// Mitsubishi GX Works2 project: TEACH 실습 예제   PLC: Q03UDV

PROGRAM MAIN
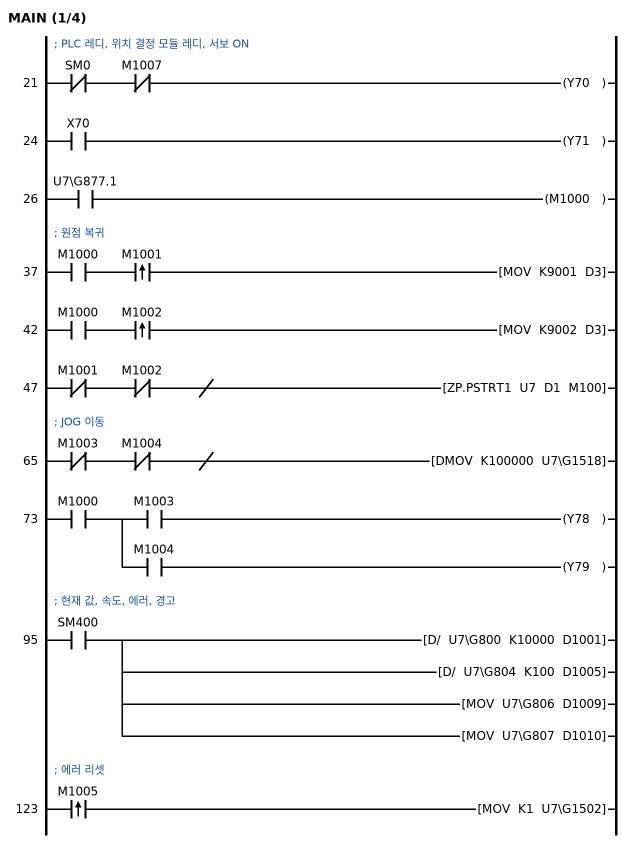
; PLC 레디, 위치 결정 모듈 레디, 서보 ON
21    LDI     SM0
      ANI     M1007
      OUT     Y70
24    LD      X70
      OUT     Y71
26    LD      U7\G877.1
      OUT     M1000
; 원점 복귀
37    LD      M1000
      ANDP    M1001
      MOV     K9001 D3
42    LD      M1000
      ANDP    M1002
      MOV     K9002 D3
47    LDI     M1001
      ANI     M1002
      INV
      ZP.PSTRT1 U7 D1 M100
; JOG 이동
65    LDI     M1003
      ANI     M1004
      INV
      DMOV    K100000 U7\G1518
73    LD      M1000
      MPS
      AND     M1003
      OUT     Y78
      MPP
      AND     M1004
      OUT     Y79
; 현재 값, 속도, 에러, 경고
95    LD      SM400
      D/      U7\G800 K10000 D1001
      D/      U7\G804 K100 D1005
      MOV     U7\G806 D1009
      MOV     U7\G807 D1010
; 에러 리셋
123   LDP     M1005
      MOV     K1 U7\G1502
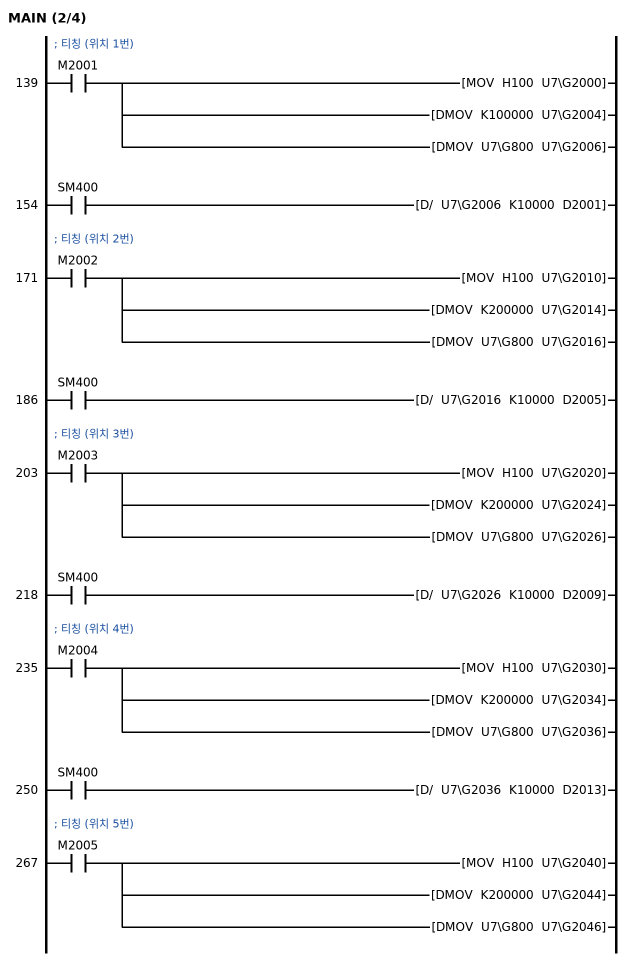
; 티칭 (위치 1번)
139   LD      M2001
      MOV     H100 U7\G2000
      DMOV    K100000 U7\G2004
      DMOV    U7\G800 U7\G2006
154   LD      SM400
      D/      U7\G2006 K10000 D2001
; 티칭 (위치 2번)
171   LD      M2002
      MOV     H100 U7\G2010
      DMOV    K200000 U7\G2014
      DMOV    U7\G800 U7\G2016
186   LD      SM400
      D/      U7\G2016 K10000 D2005
; 티칭 (위치 3번)
203   LD      M2003
      MOV     H100 U7\G2020
      DMOV    K200000 U7\G2024
      DMOV    U7\G800 U7\G2026
218   LD      SM400
      D/      U7\G2026 K10000 D2009
; 티칭 (위치 4번)
235   LD      M2004
      MOV     H100 U7\G2030
      DMOV    K200000 U7\G2034
      DMOV    U7\G800 U7\G2036
250   LD      SM400
      D/      U7\G2036 K10000 D2013
; 티칭 (위치 5번)
267   LD      M2005
      MOV     H100 U7\G2040
      DMOV    K200000 U7\G2044
      DMOV    U7\G800 U7\G2046
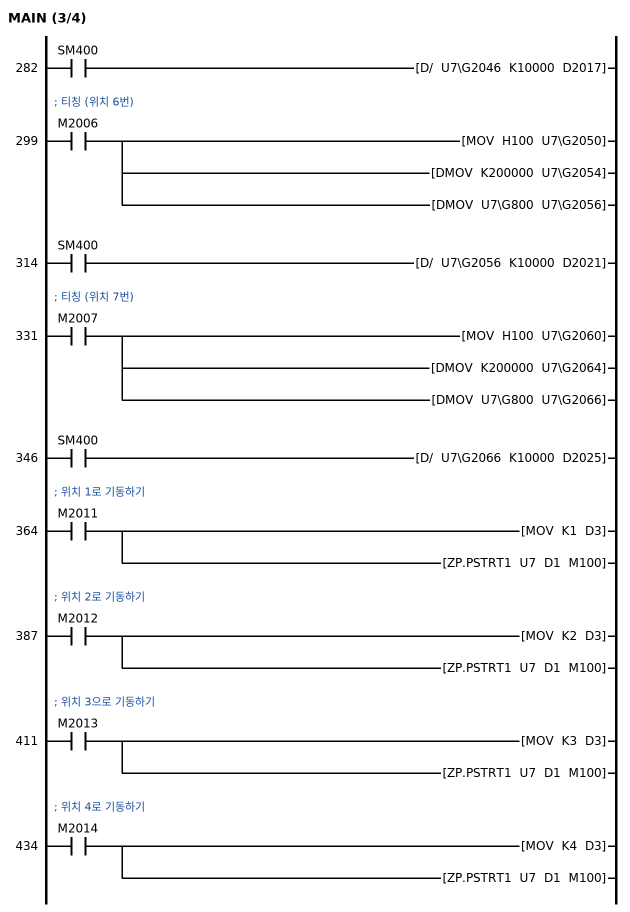
282   LD      SM400
      D/      U7\G2046 K10000 D2017
; 티칭 (위치 6번)
299   LD      M2006
      MOV     H100 U7\G2050
      DMOV    K200000 U7\G2054
      DMOV    U7\G800 U7\G2056
314   LD      SM400
      D/      U7\G2056 K10000 D2021
; 티칭 (위치 7번)
331   LD      M2007
      MOV     H100 U7\G2060
      DMOV    K200000 U7\G2064
      DMOV    U7\G800 U7\G2066
346   LD      SM400
      D/      U7\G2066 K10000 D2025
; 위치 1로 기동하기
364   LD      M2011
      MOV     K1 D3
      ZP.PSTRT1 U7 D1 M100
; 위치 2로 기동하기
387   LD      M2012
      MOV     K2 D3
      ZP.PSTRT1 U7 D1 M100
; 위치 3으로 기동하기
411   LD      M2013
      MOV     K3 D3
      ZP.PSTRT1 U7 D1 M100
; 위치 4로 기동하기
434   LD      M2014
      MOV     K4 D3
      ZP.PSTRT1 U7 D1 M100
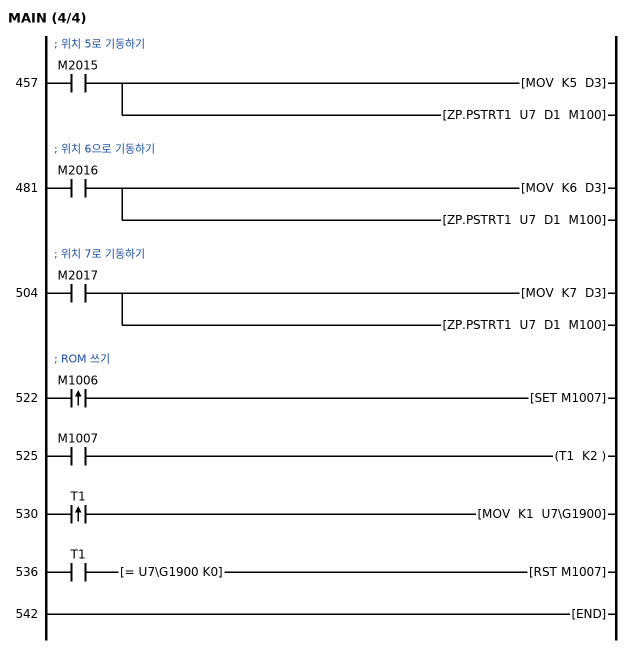
; 위치 5로 기동하기
457   LD      M2015
      MOV     K5 D3
      ZP.PSTRT1 U7 D1 M100
; 위치 6으로 기동하기
481   LD      M2016
      MOV     K6 D3
      ZP.PSTRT1 U7 D1 M100
; 위치 7로 기동하기
504   LD      M2017
      MOV     K7 D3
      ZP.PSTRT1 U7 D1 M100
; ROM 쓰기
522   LDP     M1006
      SET     M1007
525   LD      M1007
      OUT     T1 K2
530   LDP     T1
      MOV     K1 U7\G1900
536   LD      T1
      AND=    U7\G1900 K0
      RST     M1007
542   END
END_PROGRAM
